TYPE ST_PNInput_DCBusExpansion :
STRUCT
	ControlBits	:	DWORD;
END_STRUCT
END_TYPE

(* stored: Version 1.1.0.1, ProductVersion 3.1.4024.12
   DUT ST_PNInput_DCBusExpansion: Id {5be21798-600a-4ffb-bf70-d3f3d3ddadb0} *)
